// ==============================================================================
// DB_IO_Config_Doc
// Документація конфігурації I/O мапінгу
//
// Згенеровано автоматично: 2026-01-13 16:47:15
// Джерело: IO_Config.xlsx
// Механізмів: 2
// ==============================================================================

DATA_BLOCK "DB_IO_Config_Doc"
{ S7_Optimized_Access := 'TRUE' }

VAR
    // Налаштування HAL
    HAL_Enabled    : BOOL := TRUE;   // увімкнути HAL
    HAL_SafeMode   : BOOL := FALSE;  // safe mode = всі виходи OFF
    HAL_DiagMode   : BOOL := FALSE;  // діагностичний режим

    // Статистика
    HAL_ReadCycles  : UDINT;  // лічильник циклів READ
    HAL_WriteCycles : UDINT;  // лічильник циклів WRITE
    HAL_Errors      : UINT;   // лічильник помилок

    // Конфігурація проекту
    TotalMechanisms : UINT := 2;
    ConfigSource    : STRING[64] := 'IO_Config.xlsx';
END_VAR

BEGIN
    // ==========================================================================
    // МАПІНГ МЕХАНІЗМІВ (для документації)
    // ==========================================================================
    //
    // Slot 0: TypedIndex 0
    // Name: Redler_Intake_1
    // Comment: Прийом зерна
    // Inputs:  %I0.0, %I0.1, %I0.2
    // Output:  %Q0.0
    //
    // Slot 1: TypedIndex 1
    // Name: Redler_Tower_B2
    // Comment: Вежа Б2
    // Inputs:  %I0.3, %I0.4, %I0.5
    // Output:  %Q0.1
    // Inverted: Breaker

END_DATA_BLOCK